PROGRAM MAIN
VAR
	fbFMS205 : L6_FMS205;	
END_VAR

fbFMS205.ProcessCycle();

END_PROGRAM

(* stored: Version 1.1.0.1, ProductVersion 3.1.4024.11
   POU MAIN: Id {19798f55-9da0-48b7-a2d0-4bd977cab0f2}, SpecialFunc None *)
